Staubli VAL3: control.pgx

public program control()
begin
  //
  // use to check your own task create in the OnStartup program
  //
end
